{attribute 'GeneratedUsingTerminal: EK1960-0000-0019'}
{attribute addProperty BoxType "EK1960-0000-0019"}
{attribute addProperty Id "FSOEAT %Q*FSOE_BAC7BF2151"}
{attribute addProperty CRC "2045205931"}
{attribute addProperty Size "51"}
TYPE FSoE_Outputs_79E75DAB EXTENDS OutputBase_10CEE7DE :
STRUCT
	{attribute addProperty Name "FSOE"}
	FSOE AT %Q* : FSOE_BAC7BF21;
END_STRUCT
END_TYPE

(* stored: Version 1.2.0.0, ProductVersion 3.1.4024.11
   DUT FSoE_Outputs_79E75DAB: Id {eefa0631-6ed8-4ec3-b4ef-b3ee1f00444f} *)
